FUNCTION_BLOCK BallSeatStation EXTENDS MachineStation
VAR_INPUT
	rIO				: REFERENCE TO BallSeat_IO_typ;
	rStation		: REFERENCE TO Station;
	rPrintStation	: REFERENCE TO MultiStation;
END_VAR
VAR_OUTPUT
END_VAR
VAR
	test:INT;
	Payload	: Payload_typ;
END_VAR

IF NOT (__ISVALIDREF(rStation) AND __ISVALIDREF(rIO) AND __ISVALIDREF(rPrintStation)) THEN
	ADSLOGSTR( ADSLOG_MSGTYPE_ERROR, 'Invalid reference at %s.', InstancePath);	// how to make this work?
	RETURN;
END_IF

// WHATS THE DIFFERENCE BETWEEN PUTTING THIS HERE VS FB.Cyclic Method?

IF Enable THEN
	IF NOT _Enable THEN
		;
	END_IF

	CASE State OF
		STN_WAIT:
			IF Run AND rStation.MoverInPosition THEN
				Payload						:= rStation.CurrentMover.Payload;
				rIO.Outputs.BallClampOpen	:= TRUE;
				State						:= STN_OPENBALLCLAMP;
			END_IF

		STN_OPENBALLCLAMP:
			IF rIO.Inputs.BallClampOpened THEN
				rIO.Outputs.BallClampOpen		:= FALSE;
				rIO.Outputs.ExtendBallSeater	:= TRUE;
				State							:= STN_PROCESS;
			END_IF

		STN_PROCESS:
			IF rIO.Inputs.BallSeatExtended THEN
				rIO.Outputs.ExtendBallSeater	:= FALSE;
				rIO.Outputs.RetractBallSeater	:= TRUE;
				Payload.BallSeated				:= TRUE;
				rIO.Outputs.BallClampClose		:= TRUE;
				State							:= STN_CLOSEBALLCLAMP;
			END_IF

		STN_CLOSEBALLCLAMP:
			IF rIO.Inputs.BallClampClosed AND rIO.Inputs.BallSeatRetracted THEN
				rIO.Outputs.RetractBallSeater	:= FALSE;
				rIO.Outputs.BallClampClose		:= FALSE;
				State							:= STN_SEND;
			END_IF

		STN_SEND:
			(*IF Test = 4 THEN Payload.Reject	:= TRUE; END_IF	// TEMP - TO TEST PRINT STATION REJECT HANDLING
			Test := SEL(Test >= 4, Test + 1, 0);	*)

			rStation.CurrentMover.Payload	:= Payload;
			rStation.CurrentMover.MoveToMultiStation(rPrintStation);
			rStation.UnregisterCurrent();
			State							:= STN_WAIT;
		
		STN_ERROR:
	
	END_CASE

ELSIF _Enable THEN
	;
END_IF

//Save Previous Values
_Enable	:= Enable;

END_FUNCTION_BLOCK

(* stored: Version 1.1.0.1, ProductVersion 3.1.4024.12
   POU BallSeatStation: Id {b1740a50-d861-0608-1e6c-96015d42fa0c}, SpecialFunc None *)
